// TIA Portal V17 export
// export: Created 2024-10-17T14:16:15.5915978Z, ExportSetting WithDefaults, DisplayName Totally Integrated Automation Portal, DisplayVersion V17 Update 4, DisplayName TIA Portal Openness, DisplayVersion V17 Update 4, DisplayName TIA Portal Version Control Interface, DisplayVersion V17, DisplayName SINAMICS Startdrive Advanced, DisplayVersion V17 Update2, DisplayName SINAMICS Startdrive G130, G150, S120, S150, SINAMICS MV, S210, DisplayVersion V17 Update2, DisplayName SINAMICS Startdrive G110M, G120, G120C, G120D, G120P, G115D, DisplayVersion V17 Update2, DisplayName STEP 7 Professional, DisplayVersion V17 Update 4, DisplayName STEP 7 Safety, DisplayVersion V17, DisplayName WinCC Advanced / Unified PC, DisplayVersion V17 Update 4
DATA_BLOCK "InstLPMLV2022_UnitModeStateTimes"   // DB30112
{ DB_Accessible_From_OPC_UA := 'FALSE' }
AUTHOR : APC_ERLF
FAMILY : OMAC
VERSION : 1.0
// stored: AutoNumber true, DBAccessibleFromOPCUA false, DBAccessibleFromWebserver false, InstanceOfName LPMLV2022_UnitModeStateTimes, InstanceOfType FB
"LPMLV2022_UnitModeStateTimes"
   // VAR_INPUT
   //    UnitModeCurrent : DInt;
   //    StateCurrent : DInt;
   //    resetTimes : Bool;
   // END_VAR
   // VAR_OUTPUT
   //    ModeTimeCurrent { ExternalWritable := 'False'} : DInt;
   //    StateTimeCurrent { ExternalWritable := 'False'} : DInt;
   //    AccTimeSinceReset { ExternalWritable := 'False'} : DInt;
   //    actualTimeAllModes { ExternalWritable := 'False'} : Array[0.."LPMLV2022_MODES_UPPER_LIM"] of DInt;
   //    cumulativeTimeAllModes { ExternalWritable := 'False'} : Array[0.."LPMLV2022_MODES_UPPER_LIM"] of DInt;
   //    actualTimeAllStatesOfAllModes { ExternalWritable := 'False'} : Array[0.."LPMLV2022_MODES_UPPER_LIM", 0.."LPMLV2022_STATES_UPPER_LIM"] of DInt;
   //    cumulativeTimeAllStatesOfAllModes { ExternalWritable := 'False'} : Array[0.."LPMLV2022_MODES_UPPER_LIM", 0.."LPMLV2022_STATES_UPPER_LIM"] of DInt;
   //    actualTimeAllStatesOfCurrentMode { ExternalWritable := 'False'} : Array[0.."LPMLV2022_STATES_UPPER_LIM"] of DInt;
   //    cumulativeTimeAllStatesOfCurrentMode { ExternalWritable := 'False'} : Array[0.."LPMLV2022_STATES_UPPER_LIM"] of DInt;
   //    cumulativeTimeCurrentMode { ExternalWritable := 'False'} : DInt;
   // END_VAR
   // VAR
   //    statUnitModeCurrentOld { ExternalAccessible := 'False'; ExternalVisible := 'False'; ExternalWritable := 'False'} : DInt;
   //    statStateCurrentOld { ExternalAccessible := 'False'; ExternalVisible := 'False'; ExternalWritable := 'False'} : DInt;
   //    statResetTimesOld { ExternalAccessible := 'False'; ExternalVisible := 'False'; ExternalWritable := 'False'} : Bool;
   //    statStartingPointMeasureRuntime { ExternalAccessible := 'False'; ExternalVisible := 'False'; ExternalWritable := 'False'} : LReal;
   //    statRuntime { ExternalAccessible := 'False'; ExternalVisible := 'False'; ExternalWritable := 'False'} : LReal;
   //    statFirstCycle { ExternalAccessible := 'False'; ExternalVisible := 'False'; ExternalWritable := 'False'} : Bool;
   //    statCurrentModeCurrentTime { ExternalAccessible := 'False'; ExternalVisible := 'False'; ExternalWritable := 'False'} : DInt;
   //    statCurrentStateCurrentTime { ExternalAccessible := 'False'; ExternalVisible := 'False'; ExternalWritable := 'False'} : DInt;
   // END_VAR
BEGIN
END_DATA_BLOCK
